// TIA Portal V20 export
DATA_BLOCK "ProdDataInterfaceHmi"   // DB53
TITLE = HMI und Anwender Schnittstelle für Produktionsdaten / HMI and user interface for production data
AUTHOR : SICAR
FAMILY : ProdData
// FUNKTIONSBESCHREIBUNG: 
// Der Baustein beinhaltet alle Informationen zum und vom HMI, sowie die Anwenderschnittstellen für die Produktionsdaten
// Weitere Hinweise: siehe SICAR anwenderdefinierte Dokumentation / SICAR Online-Hilfe.
// DESCRIPTION OF FUNCTIONS:
// stored: MemoryReserve 100
   VAR RETAIN
      numberOfDataSets : "LSicar_typeNumberOfDataSets";   // Anzahl konfigurierter Datensätze / Number of configured data sets
   END_VAR
   VAR
      colorCodeLimitSummary : UInt := 0;   // Gesamt Status Grenzwerte / Overall status Limit values
      colorCodeLimitSelButton : Array[0..8] of UInt;   // Farbcode für Datensatz Anwahl Button (Grenzwerte) / Color code for data set select button (Limit values)
   END_VAR
   VAR RETAIN
      limitValueDataSetSel : Int := 1;   // Angwaehlter Datensatz Grenzwerte / selected data set limit values
      limitDataSet : Array[0.."NO_DATASETS_LIMITVALUES"] of "LSicar_typeLimitValue";   // Datensätze Grenzwerte / Data sets limit .values
      cycleTimerDataSetSel : Int := 1;   // Angewaehlter Datensatz Taktzeiten / selected data set cycle timer
      cycleTimerDataSet : Array[0.."NO_DATASETS_CYCLETIMER"] of "LSicar_typeCycleTimer";   // Datensätze Taktzeiten / Data sets cycle timer
      counterDataSetSel : Int := 1;   // Angewählter Datensatz Zaehler / selected data set counter
      counterDataSet : Array[0.."NO_DATASETS_COUNTER"] of "LSicar_typeCounter";   // Datensätze Zähler / Data sets counter
      shiftCounterDataSetSel : Int := 1;   // Angewaehlter Datensatz Schichtzaehler / selected data set shift counter
      shiftCounterDataSet : Array[0.."NO_DATASETS_SHIFTCOUNTER"] of "LSicar_typeShiftCounter";   // Datensätze Schichtzähler / Data sets shift counter
      shiftCountOeeDataSetSel : Int := 1;   // Angewaehlter Datensatz OEE / selected data set OEE
      shiftCounterOeeDataSet : Array[0.."NO_DATASETS_SHIFTCOUNTER"] of "LSicar_typeShiftCounterOee";   // Datensätze Schichtzähler OEE / Data sets shift counter OEE
   END_VAR
BEGIN
   numberOfDataSets.limitValues := 2;
   numberOfDataSets.cycleTimer := 2;
   numberOfDataSets."counter" := 2;
   numberOfDataSets.shiftCounter := 2;
   colorCodeLimitSelButton[0..8] := 0;
   limitDataSet[0].targetValue[0..10] := 0;
   limitDataSet[1].targetValue[0..10] := 0;
   limitDataSet[2].targetValue[0..10] := 0;
   limitDataSet[0].prewarnValue[0..10] := 0;
   limitDataSet[1].prewarnValue[0..10] := 0;
   limitDataSet[2].prewarnValue[0..10] := 0;
   limitDataSet[0].remainValue[0..10] := 0;
   limitDataSet[1].remainValue[0..10] := 0;
   limitDataSet[2].remainValue[0..10] := 0;
   limitDataSet[0].control[0..10].count := FALSE;
   limitDataSet[1].control[0..10].count := FALSE;
   limitDataSet[2].control[0..10].count := FALSE;
   limitDataSet[0].control[0..10].set := FALSE;
   limitDataSet[1].control[0..10].set := FALSE;
   limitDataSet[2].control[0..10].set := FALSE;
   limitDataSet[0].control[0..10].prewarn := FALSE;
   limitDataSet[1].control[0..10].prewarn := FALSE;
   limitDataSet[2].control[0..10].prewarn := FALSE;
   limitDataSet[0].control[0..10].alarm := FALSE;
   limitDataSet[1].control[0..10].alarm := FALSE;
   limitDataSet[2].control[0..10].alarm := FALSE;
   limitDataSet[0].textListValue[0..10] := 0;
   limitDataSet[1].textListValue[0..10] := 0;
   limitDataSet[2].textListValue[0..10] := 0;
   limitDataSet[0..2].userInterfaceVisibility := 16#0000_0000;
   limitDataSet[0].colorCodeAlarmPrewarn[0..10] := 0;
   limitDataSet[1].colorCodeAlarmPrewarn[0..10] := 0;
   limitDataSet[2].colorCodeAlarmPrewarn[0..10] := 0;
   limitDataSet[0..2].indexSelectedLimitValue := 0;
   limitDataSet[0..2].divButton := 16#00;
   limitDataSet[0..2].visibility := 16#0000_0000;
   cycleTimerDataSet[0].targetValue[0..20] := 0;
   cycleTimerDataSet[1].targetValue[0..20] := 0;
   cycleTimerDataSet[2].targetValue[0..20] := 0;
   cycleTimerDataSet[0].currentValue[0..20] := 0;
   cycleTimerDataSet[1].currentValue[0..20] := 0;
   cycleTimerDataSet[2].currentValue[0..20] := 0;
   cycleTimerDataSet[0].averageValue[0..20] := 0;
   cycleTimerDataSet[1].averageValue[0..20] := 0;
   cycleTimerDataSet[2].averageValue[0..20] := 0;
   cycleTimerDataSet[0].counts[0..20] := 0;
   cycleTimerDataSet[1].counts[0..20] := 0;
   cycleTimerDataSet[2].counts[0..20] := 0;
   cycleTimerDataSet[0].measureActive[0..20] := 0;
   cycleTimerDataSet[1].measureActive[0..20] := 0;
   cycleTimerDataSet[2].measureActive[0..20] := 0;
   cycleTimerDataSet[0].control[0..20].run := FALSE;
   cycleTimerDataSet[1].control[0..20].run := FALSE;
   cycleTimerDataSet[2].control[0..20].run := FALSE;
   cycleTimerDataSet[0].control[0..20].hold := FALSE;
   cycleTimerDataSet[1].control[0..20].hold := FALSE;
   cycleTimerDataSet[2].control[0..20].hold := FALSE;
   cycleTimerDataSet[0].control[0..20].reset := FALSE;
   cycleTimerDataSet[1].control[0..20].reset := FALSE;
   cycleTimerDataSet[2].control[0..20].reset := FALSE;
   cycleTimerDataSet[0].textListValue[0..20] := 0;
   cycleTimerDataSet[1].textListValue[0..20] := 0;
   cycleTimerDataSet[2].textListValue[0..20] := 0;
   cycleTimerDataSet[0..2].userInterfaceVisibility := 16#0000_0000;
   cycleTimerDataSet[0..2].resetAverageAllExt := FALSE;
   cycleTimerDataSet[0..2].indexSelectedTimer := 0;
   cycleTimerDataSet[0..2].divButton := 16#00;
   cycleTimerDataSet[0..2].visibility := 16#0000_0000;
   counterDataSet[0].currentValue[0..20] := 0;
   counterDataSet[1].currentValue[0..20] := 0;
   counterDataSet[2].currentValue[0..20] := 0;
   counterDataSet[0].control[0..20].countUp := FALSE;
   counterDataSet[1].control[0..20].countUp := FALSE;
   counterDataSet[2].control[0..20].countUp := FALSE;
   counterDataSet[0].control[0..20].countDown := FALSE;
   counterDataSet[1].control[0..20].countDown := FALSE;
   counterDataSet[2].control[0..20].countDown := FALSE;
   counterDataSet[0].control[0..20].reset := FALSE;
   counterDataSet[1].control[0..20].reset := FALSE;
   counterDataSet[2].control[0..20].reset := FALSE;
   counterDataSet[0].textListValue[0..20] := 0;
   counterDataSet[1].textListValue[0..20] := 0;
   counterDataSet[2].textListValue[0..20] := 0;
   counterDataSet[0].userInterfaceVisibility := 16#0000_0000;
   counterDataSet[1].userInterfaceVisibility := 16#0000_0007;
   counterDataSet[2].userInterfaceVisibility := 16#0000_0003;
   counterDataSet[0..2].resetAllExt := FALSE;
   counterDataSet[0..2].indexSelectedCounter := 0;
   counterDataSet[0..2].divButton := 16#00;
   counterDataSet[0..2].visibility := 16#0000_0000;
   shiftCounterDataSet[0].currentShiftValue.partsTarget[0..10] := 0;
   shiftCounterDataSet[1].currentShiftValue.partsTarget[0..10] := 0;
   shiftCounterDataSet[2].currentShiftValue.partsTarget[0..10] := 0;
   shiftCounterDataSet[0].currentShiftValue.partsCurrent[0..10] := 0;
   shiftCounterDataSet[1].currentShiftValue.partsCurrent[0..10] := 0;
   shiftCounterDataSet[2].currentShiftValue.partsCurrent[0..10] := 0;
   shiftCounterDataSet[0].previousShiftValue.partsTarget[0..10] := 0;
   shiftCounterDataSet[1].previousShiftValue.partsTarget[0..10] := 0;
   shiftCounterDataSet[2].previousShiftValue.partsTarget[0..10] := 0;
   shiftCounterDataSet[0].previousShiftValue.partsCurrent[0..10] := 0;
   shiftCounterDataSet[1].previousShiftValue.partsCurrent[0..10] := 0;
   shiftCounterDataSet[2].previousShiftValue.partsCurrent[0..10] := 0;
   shiftCounterDataSet[0].penultimateShiftValue.partsTarget[0..10] := 0;
   shiftCounterDataSet[1].penultimateShiftValue.partsTarget[0..10] := 0;
   shiftCounterDataSet[2].penultimateShiftValue.partsTarget[0..10] := 0;
   shiftCounterDataSet[0].penultimateShiftValue.partsCurrent[0..10] := 0;
   shiftCounterDataSet[1].penultimateShiftValue.partsCurrent[0..10] := 0;
   shiftCounterDataSet[2].penultimateShiftValue.partsCurrent[0..10] := 0;
   shiftCounterDataSet[0].countPartsCurrent[0..10] := FALSE;
   shiftCounterDataSet[1].countPartsCurrent[0..10] := FALSE;
   shiftCounterDataSet[2].countPartsCurrent[0..10] := FALSE;
   shiftCounterDataSet[0].textListValue[0..10] := 0;
   shiftCounterDataSet[1].textListValue[0..10] := 0;
   shiftCounterDataSet[2].textListValue[0..10] := 0;
   shiftCounterDataSet[0..2].userInterfaceVisibility := 16#0000_0000;
   shiftCounterDataSet[0..2].resetAllExt := FALSE;
   shiftCounterDataSet[0..2].divButton := 16#00;
   shiftCounterDataSet[0..2].visibility := 16#0000_0000;
   shiftCounterOeeDataSet[0].currentShiftValue.oee[0..10] := 0.0;
   shiftCounterOeeDataSet[1].currentShiftValue.oee[0..10] := 0.0;
   shiftCounterOeeDataSet[2].currentShiftValue.oee[0..10] := 0.0;
   shiftCounterOeeDataSet[0].currentShiftValue.trend[0..10] := 0;
   shiftCounterOeeDataSet[1].currentShiftValue.trend[0..10] := 0;
   shiftCounterOeeDataSet[2].currentShiftValue.trend[0..10] := 0;
   shiftCounterOeeDataSet[0].currentShiftValue.partsTarget[0..10] := 0;
   shiftCounterOeeDataSet[1].currentShiftValue.partsTarget[0..10] := 0;
   shiftCounterOeeDataSet[2].currentShiftValue.partsTarget[0..10] := 0;
   shiftCounterOeeDataSet[0].currentShiftValue.partsCurrent[0..10] := 0;
   shiftCounterOeeDataSet[1].currentShiftValue.partsCurrent[0..10] := 0;
   shiftCounterOeeDataSet[2].currentShiftValue.partsCurrent[0..10] := 0;
   shiftCounterOeeDataSet[0].currentShiftValue.partsCurrentOk[0..10] := 0;
   shiftCounterOeeDataSet[1].currentShiftValue.partsCurrentOk[0..10] := 0;
   shiftCounterOeeDataSet[2].currentShiftValue.partsCurrentOk[0..10] := 0;
   shiftCounterOeeDataSet[0].previousShiftValue.oee[0..10] := 0.0;
   shiftCounterOeeDataSet[1].previousShiftValue.oee[0..10] := 0.0;
   shiftCounterOeeDataSet[2].previousShiftValue.oee[0..10] := 0.0;
   shiftCounterOeeDataSet[0].previousShiftValue.trend[0..10] := 0;
   shiftCounterOeeDataSet[1].previousShiftValue.trend[0..10] := 0;
   shiftCounterOeeDataSet[2].previousShiftValue.trend[0..10] := 0;
   shiftCounterOeeDataSet[0].previousShiftValue.partsTarget[0..10] := 0;
   shiftCounterOeeDataSet[1].previousShiftValue.partsTarget[0..10] := 0;
   shiftCounterOeeDataSet[2].previousShiftValue.partsTarget[0..10] := 0;
   shiftCounterOeeDataSet[0].previousShiftValue.partsCurrent[0..10] := 0;
   shiftCounterOeeDataSet[1].previousShiftValue.partsCurrent[0..10] := 0;
   shiftCounterOeeDataSet[2].previousShiftValue.partsCurrent[0..10] := 0;
   shiftCounterOeeDataSet[0].previousShiftValue.partsCurrentOk[0..10] := 0;
   shiftCounterOeeDataSet[1].previousShiftValue.partsCurrentOk[0..10] := 0;
   shiftCounterOeeDataSet[2].previousShiftValue.partsCurrentOk[0..10] := 0;
   shiftCounterOeeDataSet[0].penultimateShiftValue.oee[0..10] := 0.0;
   shiftCounterOeeDataSet[1].penultimateShiftValue.oee[0..10] := 0.0;
   shiftCounterOeeDataSet[2].penultimateShiftValue.oee[0..10] := 0.0;
   shiftCounterOeeDataSet[0].penultimateShiftValue.trend[0..10] := 0;
   shiftCounterOeeDataSet[1].penultimateShiftValue.trend[0..10] := 0;
   shiftCounterOeeDataSet[2].penultimateShiftValue.trend[0..10] := 0;
   shiftCounterOeeDataSet[0].penultimateShiftValue.partsTarget[0..10] := 0;
   shiftCounterOeeDataSet[1].penultimateShiftValue.partsTarget[0..10] := 0;
   shiftCounterOeeDataSet[2].penultimateShiftValue.partsTarget[0..10] := 0;
   shiftCounterOeeDataSet[0].penultimateShiftValue.partsCurrent[0..10] := 0;
   shiftCounterOeeDataSet[1].penultimateShiftValue.partsCurrent[0..10] := 0;
   shiftCounterOeeDataSet[2].penultimateShiftValue.partsCurrent[0..10] := 0;
   shiftCounterOeeDataSet[0].penultimateShiftValue.partsCurrentOk[0..10] := 0;
   shiftCounterOeeDataSet[1].penultimateShiftValue.partsCurrentOk[0..10] := 0;
   shiftCounterOeeDataSet[2].penultimateShiftValue.partsCurrentOk[0..10] := 0;
   shiftCounterOeeDataSet[0].countPartsCurrent[0..10] := FALSE;
   shiftCounterOeeDataSet[1].countPartsCurrent[0..10] := FALSE;
   shiftCounterOeeDataSet[2].countPartsCurrent[0..10] := FALSE;
   shiftCounterOeeDataSet[0].countPartsCurrentOk[0..10] := FALSE;
   shiftCounterOeeDataSet[1].countPartsCurrentOk[0..10] := FALSE;
   shiftCounterOeeDataSet[2].countPartsCurrentOk[0..10] := FALSE;
   shiftCounterOeeDataSet[0].textListValue[0..10] := 0;
   shiftCounterOeeDataSet[1].textListValue[0..10] := 0;
   shiftCounterOeeDataSet[2].textListValue[0..10] := 0;
   shiftCounterOeeDataSet[0..2].userInterfaceVisibility := 16#0000_0000;
   shiftCounterOeeDataSet[0..2].resetAllExt := FALSE;
   shiftCounterOeeDataSet[0..2].divButton := 16#00;
   shiftCounterOeeDataSet[0..2].visibility := 16#0000_0000;
END_DATA_BLOCK
